(* IEC 61131-3 sources: axftcmlib/src/Compressor, 4 files *)

(* ---- IPneumaticCompressor.st ---- *)
NAMESPACE Simatic.Ax.axftcmlib
INTERFACE IPneumaticCompressor

        METHOD PneumaticCompressorOn
        END_METHOD
        METHOD PneumaticCompressorOff
        END_METHOD
    END_INTERFACE

END_NAMESPACE

(* ---- itfPowerableDevice.st ---- *)
///Interface for a class compressor
///contains the basic functions neede for the Fischertechnik models
/// Is used to power a pneumatic cylinder
NAMESPACE Simatic.Ax.axftcmlib

    INTERFACE itfPowerableDevice
        ///turns the device on
        METHOD PowerOn
        END_METHOD
        ///turns the device off
        METHOD PowerOff
        END_METHOD
        /// Is powered On
        METHOD IsPoweredOn : BOOL
        END_METHOD
    END_INTERFACE

END_NAMESPACE

(* ---- Compressor.st ---- *)
USING Simatic.Ax.IO.Input;
USING Simatic.Ax.IO.Output;
USING Simatic.Ax.Commands;

NAMESPACE Simatic.Ax.axftcmlib

    ///Implementation of the Compressor interface
    /// needs an ItfBinOutout that is used to write on the PLC-Variables
    CLASS Compressor
        EXTENDS EnablingControlModuleAbstract
        IMPLEMENTS IEnablingCm
        VAR PUBLIC
            QControl : ItfBinOutput;
        END_VAR
        ///turns the compressor on

        METHOD PUBLIC Enable : itfCommand
            IF QControl = NULL THEN
                Enable := THIS;
                RETURN;
            END_IF;
            QControl.SetOn();
            THIS.InitState();
            Enable := THIS;
        END_METHOD
        ///turns the compressor off

        METHOD PUBLIC Disable : itfCommand
            Disable := THIS;
            IF THIS._Error THEN
                RETURN;
            END_IF;
            QControl.SetOff();
            THIS.SetDone();
        END_METHOD

        METHOD PROTECTED OVERRIDE _executeCustom
            IF THIS._Error THEN
                RETURN;
            END_IF;
            QControl.SetOn();
        END_METHOD

        METHOD PROTECTED OVERRIDE _initmethod
            IF (QControl = NULL) THEN
                THIS.SetError(WORD#16#8001);
            END_IF;
        END_METHOD
    END_CLASS

END_NAMESPACE

(* ---- PneumaticCompressor.st ---- *)
USING Simatic.Ax.IO.Input;

USING Simatic.Ax.IO.Output;
NAMESPACE Simatic.Ax.axftcmlib

    CLASS  PneumaticCompressor IMPLEMENTS  IPneumaticCompressor

        VAR PUBLIC
             ActiveCompressor : IBinOutput;
        END_VAR

        METHOD PUBLIC PneumaticCompressorOn
           ActiveCompressor.SetOn() ;
        END_METHOD

        METHOD PUBLIC PneumaticCompressorOff
            ActiveCompressor.SetOff();
        END_METHOD
    END_CLASS

END_NAMESPACE
